Staubli VAL3: loadPage.pgx

program loadPage(string x_sPage (dimensions=1), string& x_sItems[] (dimensions=1))
// load the next page
  local num i
begin
  // look if the page libload is correct
  i=page:libLoad(x_sPage)
  if i!=0
    logMsg("[VALPLAST] INTERFACE:PAGE LIBLOAD "+x_sPage+" result "+toString("",i))
    popUpMsg("Loading page "+x_sPage+" error CODE "+toString("",i))
  else
    // copy all the field from x_sItems to the next page
    page:sItems=x_sItems
    call page:main()
    // to give back
    x_sItems=page:sItems
  endIf
end
